Yaskawa INFORM job: SQUARE.JBI

/JOB
//NAME SQUARE
//POS
///NPOS 5,0,0,0,0,0
///TOOL 0
///POSTYPE PULSE
///PULSE
C00000=0,0,0,0,0,0
C00001=20000,0,0,0,0,0
C00002=20000,20000,0,0,0,0
C00003=0,20000,0,0,0,0
C00004=0,0,0,0,0,0
//INST
///DATE 2026/04/01 12:00
///ATTR SC,RW
///GROUP1 RB1
NOP
MOVJ C00000 VJ=25.00
MOVL C00001 V=200.0
MOVL C00002 V=200.0
MOVL C00003 V=200.0
MOVL C00004 V=200.0
END
